{attribute addProperty BoxType "AX8118-0000-0100-0100"}
{attribute addProperty Id "DeviceDevice_F82A60211620Ch_ACh_A_359CD49A176220WcStateAT %I*WcState_F855686C1620InfoDataAT %I*InfoData_F030DC9B200250"}
{attribute addProperty CRC "4200169757"}
{attribute addProperty SizeInBites "408"}
{attribute addProperty SizeInBytes "51"}
TYPE AX8118_D97ACBDE :
STRUCT
	{attribute addProperty Name "Device"}
	Device : Device_F82A6021;
	{attribute addProperty Name "Ch_A"}
	Ch_A : Ch_A_359CD49A;
	{attribute addProperty Name "WcState"}
	WcState : WcState_F855686C;
	{attribute addProperty Name "InfoData"}
	InfoData : InfoData_F030DC9B;
END_STRUCT
END_TYPE

(* stored: Version 1.2.0.0, ProductVersion 3.1.4024.9
   DUT AX8118_D97ACBDE: Id {4d0e83c4-ac02-46f7-86da-c5a7f2342600} *)
